(* Logix 5000 project; controller DAD143_Test0 1769-L16ER-BB1B rev 34.12; software revision 34.01 *)

TASK MainTask (continuous, watchdog 500 ms) : MainProgram

MODULES
   Local : 1769-L16ER-BB1B (PointIO 0, rev 34.12)
      DAD143_1 : vendor 1358 type 12 code 1430 (Ethernet 192.168.210.10, rev 1.4, StandardDataDriven RPI 20 ms)
      Discrete_IO : Embedded (PointIO 1, rev 34.11, Output RPI 20 ms)
END_MODULES

ADD_ON_INSTRUCTION AOI_DAD_143_Read   (* revision 1.0 *)
VAR_INPUT
   Index_0 : SINT; {visible}
   Index_1 : SINT; {visible}
   Subindex : SINT; {visible}
END_VAR
VAR_IN_OUT
   Out_Parameter : SINT[3]; {required}
END_VAR

ROUTINE Logic   (* ladder *)
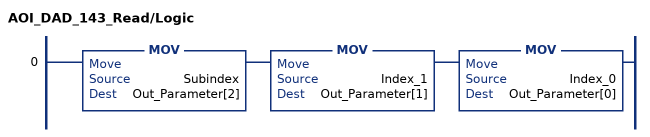
   0: MOV(Subindex,Out_Parameter[2])MOV(Index_1,Out_Parameter[1])MOV(Index_0,Out_Parameter[0]);
END_ROUTINE
END_ADD_ON_INSTRUCTION

ADD_ON_INSTRUCTION AOI_DAD_143_Write   (* revision 1.0 *)
VAR_IN_OUT
   Index_and_Subindex : SINT[3]; {required}
END_VAR
VAR_INPUT
   Data_0 : SINT; {required}
   Data_1 : SINT; {required}
   Data_2 : SINT; {required}
   Data_3 : SINT; {required}
END_VAR
VAR_IN_OUT
   Write_Par : SINT[7]; {required}
END_VAR

ROUTINE Logic   (* ladder *)
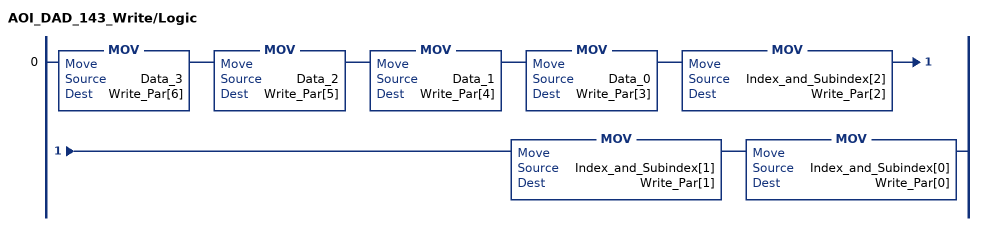
   0: MOV(Data_3,Write_Par[6])MOV(Data_2,Write_Par[5])MOV(Data_1,Write_Par[4])MOV(Data_0,Write_Par[3])MOV(Index_and_Subindex[2],Write_Par[2])MOV(Index_and_Subindex[1],Write_Par[1])MOV(Index_and_Subindex[0],Write_Par[0]);
END_ROUTINE
END_ADD_ON_INSTRUCTION

ADD_ON_INSTRUCTION AOI_DAD_143_Write_1   (* revision 1.0 *)
VAR_INPUT
   Index_0 : SINT; {visible}
   Index_1 : SINT; {visible}
   Subindex : SINT; {visible}
   Data_0 : SINT; {visible}
   Data_1 : SINT; {visible}
   Data_2 : SINT; {visible}
   Data_3 : SINT; {visible}
END_VAR
VAR_IN_OUT
   Write_Par : SINT[7]; {required}
END_VAR

ROUTINE Logic   (* ladder *)
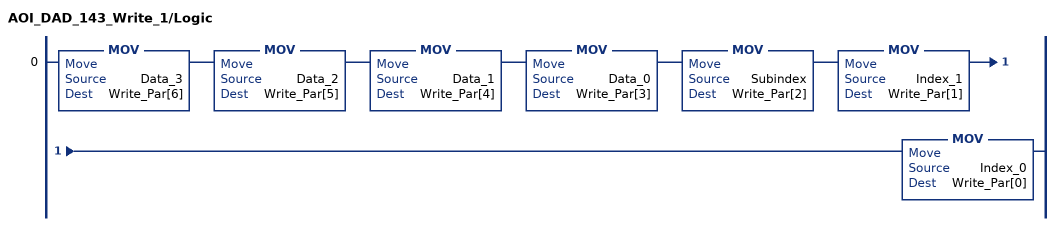
   0: MOV(Data_3,Write_Par[6])MOV(Data_2,Write_Par[5])MOV(Data_1,Write_Par[4])MOV(Data_0,Write_Par[3])MOV(Subindex,Write_Par[2])MOV(Index_1,Write_Par[1])MOV(Index_0,Write_Par[0]);
END_ROUTINE
END_ADD_ON_INSTRUCTION

VAR_GLOBAL   (* controller tags *)
   CE_Read : BOOL;
   CE_Read_Par : SINT[3];
   CE_Read_Res : SINT[5] := ([0] := 16#0b);
   CE_Read_Value : SINT := 11;
   CE_Read_Value_1 : SINT;
   CE_Read_Value_2 : SINT;
   CE_Read_Value_3 : SINT;
   CE_Start : BOOL;
   CE_Step1 : BOOL;
   CE_Step2 : BOOL;
   CE_Step3 : BOOL;
   CE_Write : BOOL;
   CI_Change : BOOL;
   CI_Change_Handshake : BOOL;
   CI_Change_Tag : BOOL;
   CI_Read_Par : SINT[3];
   CI_Step1 : BOOL;
   CI_Val : DINT;
   CM1_Change : BOOL;
   CM1_Change_Handshake : BOOL;
   CM1_Change_Tag : BOOL;
   CM1_Read_Par : SINT[3];
   CM1_Step1 : BOOL;
   CM1_Val : DINT;
   CM2_Change : BOOL;
   CM2_Change_Handshake : BOOL;
   CM2_Change_Tag : BOOL;
   CM2_Read_Par : SINT[3];
   CM2_Step1 : BOOL;
   CM2_Val : DINT;
   CM3_Change : BOOL;
   CM3_Change_Handshake : BOOL;
   CM3_Change_Tag : BOOL;
   CM3_Read_Par : SINT[3];
   CM3_Step1 : BOOL;
   CM3_Val : DINT;
   CS_Change : BOOL;
   CS_Change_Handshake : BOOL;
   CS_Change_Tag : BOOL;
   CS_Read_Par : SINT[3];
   CS_Step1 : BOOL;
   Cycle_Start : BOOL;
   DecimalPoint : SINT;
   Display_real : REAL := 7.79;
   DisplayStr : STRING := '7.82000017';
   DP : BOOL;
   DP_Cahr : STRING := '.';
   DP_Change : BOOL;
   DP_Change_1 : BOOL;
   DP_Change_Handshake : BOOL;
   DP_Change_Tag : BOOL;
   DP_Read : BOOL;
   DP_Read_Par : SINT[3];
   DP_Read_Res : SINT[5];
   DP_Step1 : BOOL;
   DP_Val : SINT;
   DP_Write : BOOL;
   DpPos : DINT := 4;
   DS : BOOL;
   DS_Change : BOOL;
   DS_Change_Handshake : BOOL;
   DS_Change_Tag : BOOL;
   DS_Read_Par : SINT[3];
   DS_Read_Res : SINT[5];
   DS_Step1 : BOOL;
   DS_Val : DINT;
   FinalStr : STRING := '7.76';
   FM_Change : BOOL;
   FM_Change_Handshake : BOOL;
   FM_Change_Tag : BOOL;
   FM_Read_Par : SINT[3];
   FM_Step1 : BOOL;
   FM_Val : SINT;
   gross : BOOL := 1;
   Gross_Display : DINT;
   Gross_weight : BOOL := 1;
   Int_reading : BOOL;
   MR : BOOL;
   MR_Change : BOOL;
   MR_Change_Handshake : BOOL;
   MR_Change_Tag : BOOL;
   MR_Read_Par : SINT[3];
   MR_Step1 : BOOL;
   MR_Val : SINT;
   ons_1 : BOOL;
   ons_2 : BOOL;
   Power_T : TIMER[12] := ([0].PRE := 50, [1].PRE := 50, [2].PRE := 2000, [3].PRE := 50);
   Power_T0 : TIMER := (PRE := 5000);
   READ_AOI : AOI_DAD_143_Read[18] := ([0].Index_1 := 16#23, [0].Subindex := 16#03, [1].Index_1 := 16#23, [1].Subindex := 16#03, [2].Index_1 := 16#23, [2].Subindex := 16#0b, [3].Index_1 := 16#23, [3].Subindex := 16#0b, [4].Index_1 := 16#23, [4].Subindex := 16#0c, [5].Index_1 := 16#23, [5].Subindex := 16#0d, [6].Index_1 := 16#23, [6].Subindex := 16#13, [7].Index_1 := 16#23, [7].Subindex := 16#15, [8].Index_0 := 16#04, [8].Index_1 := 16#20, [8].Subindex := 16#02, [9].Index_1 := 16#23, [9].Subindex := 16#14, [10].Index_1 := 16#23, [10].Subindex := 16#07, [11].Index_1 := 16#23, [11].Subindex := 16#08, [12].Index_1 := 16#23, [12].Subindex := 16#0e, [13].Index_1 := 16#23, [13].Subindex := 16#0f, [14].Index_1 := 16#23, [14].Subindex := 16#10);
   ReadCDP : MESSAGE;
        MessageParameters(ServiceCode := 16#0032, LocalElement := DP_Read_Par[0], DestinationTag := DP_Read_Res[0], ...)
   ReadCE : MESSAGE;
        MessageParameters(ServiceCode := 16#0032, LocalElement := CE_Read_Par[0], DestinationTag := CE_Read_Res[0], ...)
   ReadDS : MESSAGE;
        MessageParameters(ServiceCode := 16#0032, LocalElement := DS_Read_Par[0], DestinationTag := DS_Read_Res[0], ...)
   Stable_Bit : BOOL := 1;
   Start : BOOL;
   Start_Visibility : BOOL;
   T10 : TIMER := (PRE := 200);
   T11 : TIMER := (PRE := 50);
   T12 : TIMER := (PRE := 200);
   T13 : TIMER := (PRE := 200);
   T14 : TIMER := (PRE := 50);
   T15 : TIMER := (PRE := 200);
   T16 : TIMER := (PRE := 200);
   T17 : TIMER := (PRE := 50);
   T18 : TIMER := (PRE := 200);
   T19 : TIMER := (PRE := 200);
   T20 : TIMER := (PRE := 50);
   T21 : TIMER := (PRE := 200);
   T22 : TIMER := (PRE := 200);
   T23 : TIMER := (PRE := 50);
   T24 : TIMER := (PRE := 200);
   T25 : TIMER := (PRE := 200);
   T26 : TIMER := (PRE := 50);
   T27 : TIMER := (PRE := 200);
   T28 : TIMER := (PRE := 200);
   T29 : TIMER := (PRE := 50);
   T30 : TIMER := (PRE := 200);
   T31 : TIMER := (PRE := 200);
   T32 : TIMER := (PRE := 50);
   T33 : TIMER := (PRE := 200);
   T34 : TIMER := (PRE := 200);
   T35 : TIMER := (PRE := 50);
   T36 : TIMER := (PRE := 200);
   T37 : TIMER := (PRE := 200);
   T38 : TIMER := (PRE := 50);
   T39 : TIMER := (PRE := 200);
   T4 : TIMER := (PRE := 200);
   T5 : TIMER := (PRE := 200);
   T6 : TIMER := (PRE := 50);
   T7 : TIMER := (PRE := 200);
   T8 : TIMER := (PRE := 50);
   T9 : TIMER := (PRE := 200);
   Tare : BOOL;
   Tare_reset : BOOL;
   Tare_Reset_1 : BOOL;
   Tare_reset_Bit : BOOL := 1;
   Tare_set : BOOL;
   Tare_set_Bit : BOOL;
   temp : BOOL;
   temp1 : BOOL;
   temp_1 : BOOL;
   TN_Change : BOOL;
   TN_Change_Handshake : BOOL;
   TN_Change_Tag : BOOL;
   TN_Read_Par : SINT[3];
   TN_Step1 : BOOL;
   TN_Val : SINT;
   Write_AOI : AOI_DAD_143_Write[12];
   Write_AOI_1 : AOI_DAD_143_Write_1[20] := ([0].Index_1 := 16#23, [0].Subindex := 16#0b, [0].Data_0 := 16#03);
   Write_CE_Par : SINT[7] := ([1] := 23, [2] := 3, [3] := 11);
   Write_CE_Status : SINT[7] := ([0] := 1);
   Write_CI_Par : SINT[7];
   Write_CI_Status : SINT[7];
   Write_CM1_Par : SINT[7];
   Write_CM1_Status : SINT[7];
   Write_CM2_Par : SINT[7];
   Write_CM2_Status : SINT[7];
   Write_CM3_Par : SINT[7];
   Write_CM3_Status : SINT[7];
   Write_CS_Par : SINT[7];
   Write_CS_Status : SINT[7];
   Write_DP_Par : SINT[7];
   Write_DP_Status : SINT[7];
   Write_DS_Par : SINT[7];
   Write_DS_Status : SINT[7];
   Write_FM_Par : SINT[7];
   Write_FM_Status : SINT[7];
   Write_MR_Par : SINT[7];
   Write_MR_Status : SINT[7];
   Write_TN_Par : SINT[7];
   Write_TN_Status : SINT[7];
   Write_ZI_Par : SINT[7];
   Write_ZI_Status : SINT[7];
   Write_ZN_Par : SINT[7];
   Write_ZN_Status : SINT[7];
   WriteCE : MESSAGE;
        MessageParameters(ServiceCode := 16#0033, LocalElement := Write_CE_Par[0], DestinationTag := Write_CE_Status[0], ...)
   WriteCI : MESSAGE;
        MessageParameters(ServiceCode := 16#0033, LocalElement := Write_CI_Par[0], DestinationTag := Write_CI_Status[0], ...)
   WriteCM1 : MESSAGE;
        MessageParameters(ServiceCode := 16#0033, LocalElement := Write_CM1_Par[0], DestinationTag := Write_CM1_Status[0], ...)
   WriteCM2 : MESSAGE;
        MessageParameters(ServiceCode := 16#0033, LocalElement := Write_CM2_Par[0], DestinationTag := Write_CM2_Status[0], ...)
   WriteCM3 : MESSAGE;
        MessageParameters(ServiceCode := 16#0033, LocalElement := Write_CM3_Par[0], DestinationTag := Write_CM3_Status[0], ...)
   WriteCS : MESSAGE;
        MessageParameters(ServiceCode := 16#0033, LocalElement := Write_CS_Par[0], DestinationTag := Write_CS_Status[0], ...)
   WriteDP : MESSAGE;
        MessageParameters(ServiceCode := 16#0033, LocalElement := Write_DP_Par[0], DestinationTag := Write_DP_Status[0], ...)
   WriteDS : MESSAGE;
        MessageParameters(ServiceCode := 16#0033, LocalElement := Write_DS_Par[0], DestinationTag := Write_DS_Status[0], ...)
   WriteFM : MESSAGE;
        MessageParameters(ServiceCode := 16#0033, LocalElement := Write_FM_Par[0], DestinationTag := Write_DS_Status[0], ...)
   WriteMR : MESSAGE;
        MessageParameters(ServiceCode := 16#0033, LocalElement := Write_MR_Par[0], DestinationTag := Write_MR_Status[0], ...)
   WriteTN : MESSAGE;
        MessageParameters(ServiceCode := 16#0033, LocalElement := Write_TN_Par[0], DestinationTag := Write_TN_Status[0], ...)
   WriteZI : MESSAGE;
        MessageParameters(ServiceCode := 16#0033, LocalElement := Write_ZI_Par[0], DestinationTag := Write_ZI_Status[0], ...)
   WriteZN : MESSAGE;
        MessageParameters(ServiceCode := 16#0033, LocalElement := Write_ZN_Par[0], DestinationTag := Write_ZN_Status[0], ...)
   Zero_reset : BOOL;
   Zero_Reset_1 : BOOL;
   Zero_reset_Bit : BOOL := 1;
   Zero_set : BOOL;
   Zero_set_Bit : BOOL;
   ZI_Change : BOOL;
   ZI_Change_Handshake : BOOL;
   ZI_Change_Tag : BOOL;
   ZI_Read_Par : SINT[3];
   ZI_Step1 : BOOL;
   ZI_Val : DINT;
   ZN_Change : BOOL;
   ZN_Change_Handshake : BOOL;
   ZN_Change_Tag : BOOL;
   ZN_Read_Par : SINT[3];
   ZN_Step1 : BOOL;
   ZN_Val : SINT;
END_VAR

PROGRAM MainProgram   (* main routine MainRoutine *)
VAR
   CE_Write_Done : BOOL;
   Done_CE : BOOL;
   DP_Change_Start : BOOL;
   T0 : TIMER := (PRE := 200);
   T1 : TIMER := (PRE := 200);
   T2 : TIMER := (PRE := 200);
   T3 : TIMER := (PRE := 200);
END_VAR

ROUTINE Calibraion_Max_1   (* ladder *)
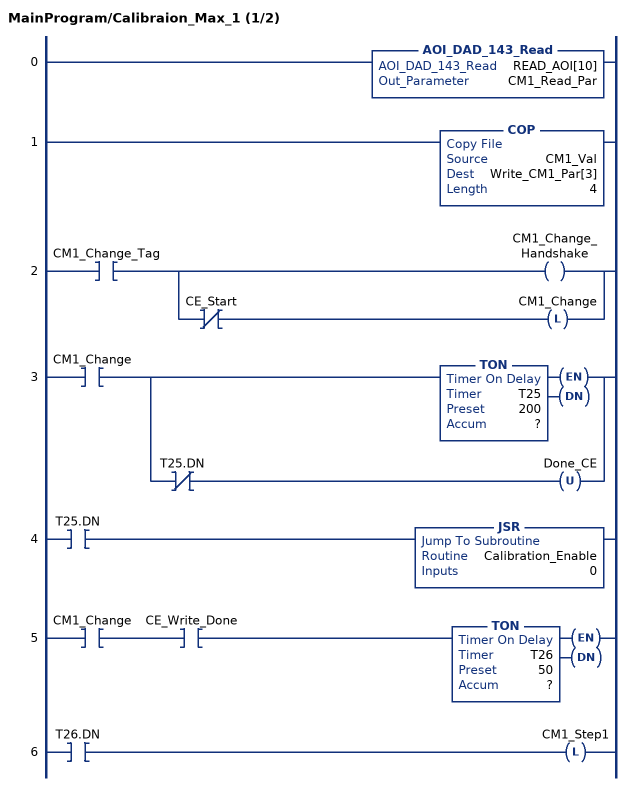
   0: AOI_DAD_143_Read(READ_AOI[10],CM1_Read_Par);
   1: COP(CM1_Val,Write_CM1_Par[3],4);
   2: XIC(CM1_Change_Tag)[OTE(CM1_Change_Handshake) ,XIO(CE_Start) OTL(CM1_Change) ];
   3: XIC(CM1_Change)[TON(T25,?,?) ,XIO(T25.DN) OTU(Done_CE) ];
   4: XIC(T25.DN)JSR(Calibration_Enable,0);
   5: XIC(CM1_Change)XIC(CE_Write_Done)TON(T26,?,?);
   6: XIC(T26.DN)OTL(CM1_Step1);
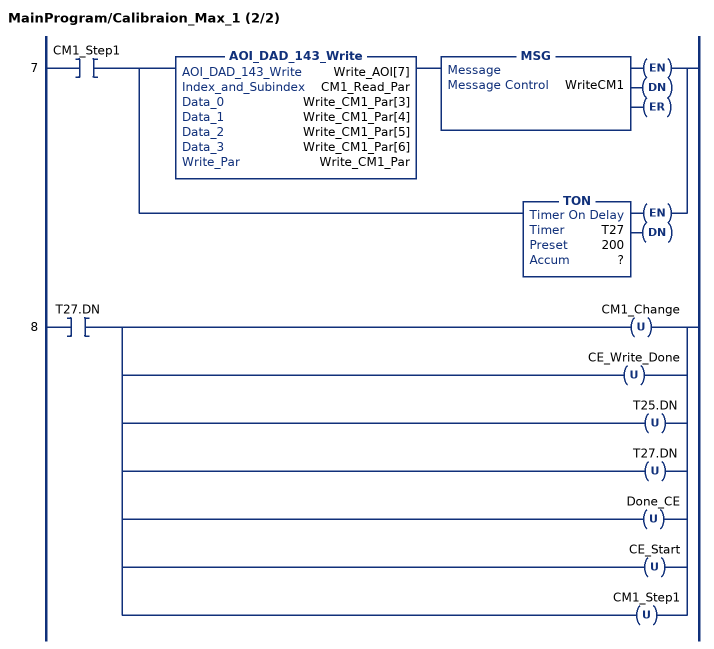
   7: XIC(CM1_Step1)[AOI_DAD_143_Write(Write_AOI[7],CM1_Read_Par,Write_CM1_Par[3],Write_CM1_Par[4],Write_CM1_Par[5],Write_CM1_Par[6],Write_CM1_Par) MSG(WriteCM1) ,TON(T27,?,?) ];
   8: XIC(T27.DN)[OTU(CM1_Change) ,OTU(CE_Write_Done) ,OTU(T25.DN) ,OTU(T27.DN) ,OTU(Done_CE) ,OTU(CE_Start) ,OTU(CM1_Step1) ];
END_ROUTINE

ROUTINE Calibraion_Max_2   (* ladder *)
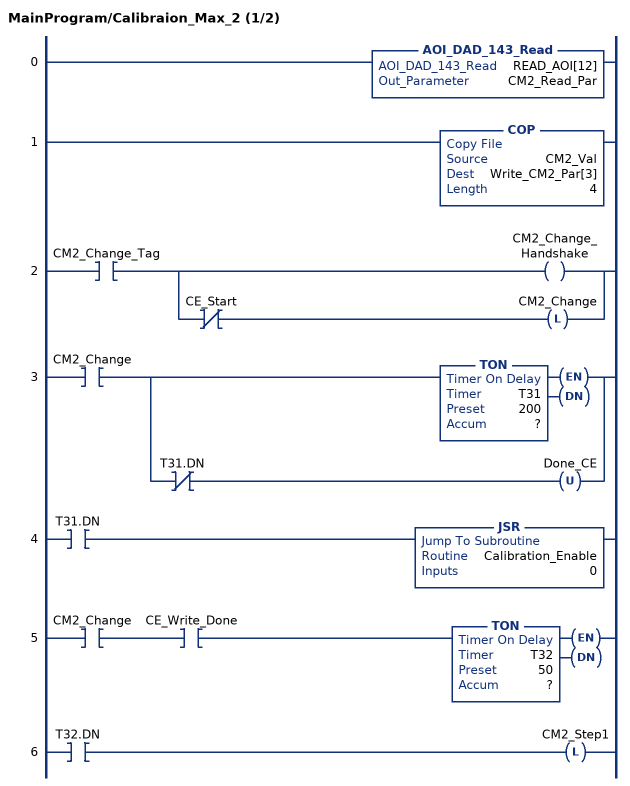
   0: AOI_DAD_143_Read(READ_AOI[12],CM2_Read_Par);
   1: COP(CM2_Val,Write_CM2_Par[3],4);
   2: XIC(CM2_Change_Tag)[OTE(CM2_Change_Handshake) ,XIO(CE_Start) OTL(CM2_Change) ];
   3: XIC(CM2_Change)[TON(T31,?,?) ,XIO(T31.DN) OTU(Done_CE) ];
   4: XIC(T31.DN)JSR(Calibration_Enable,0);
   5: XIC(CM2_Change)XIC(CE_Write_Done)TON(T32,?,?);
   6: XIC(T32.DN)OTL(CM2_Step1);
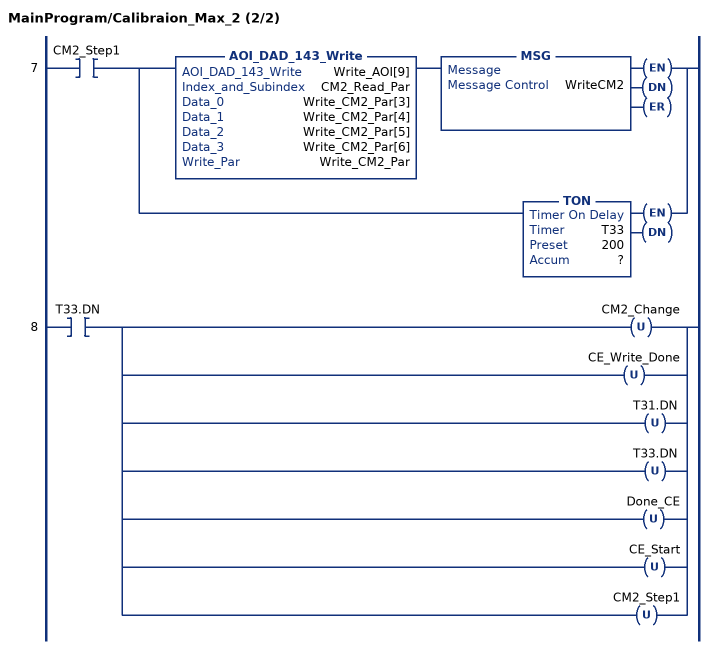
   7: XIC(CM2_Step1)[AOI_DAD_143_Write(Write_AOI[9],CM2_Read_Par,Write_CM2_Par[3],Write_CM2_Par[4],Write_CM2_Par[5],Write_CM2_Par[6],Write_CM2_Par) MSG(WriteCM2) ,TON(T33,?,?) ];
   8: XIC(T33.DN)[OTU(CM2_Change) ,OTU(CE_Write_Done) ,OTU(T31.DN) ,OTU(T33.DN) ,OTU(Done_CE) ,OTU(CE_Start) ,OTU(CM2_Step1) ];
END_ROUTINE

ROUTINE Calibraion_Max_3   (* ladder *)
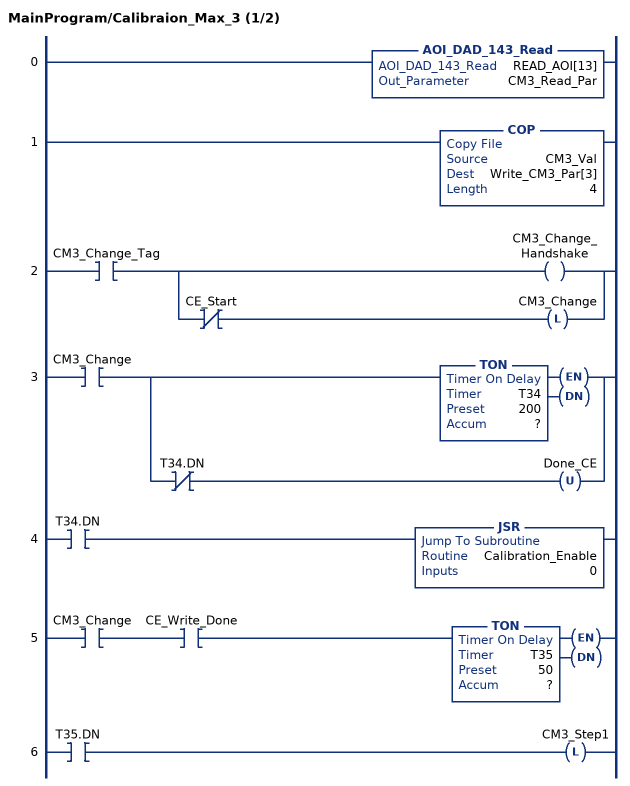
   0: AOI_DAD_143_Read(READ_AOI[13],CM3_Read_Par);
   1: COP(CM3_Val,Write_CM3_Par[3],4);
   2: XIC(CM3_Change_Tag)[OTE(CM3_Change_Handshake) ,XIO(CE_Start) OTL(CM3_Change) ];
   3: XIC(CM3_Change)[TON(T34,?,?) ,XIO(T34.DN) OTU(Done_CE) ];
   4: XIC(T34.DN)JSR(Calibration_Enable,0);
   5: XIC(CM3_Change)XIC(CE_Write_Done)TON(T35,?,?);
   6: XIC(T35.DN)OTL(CM3_Step1);
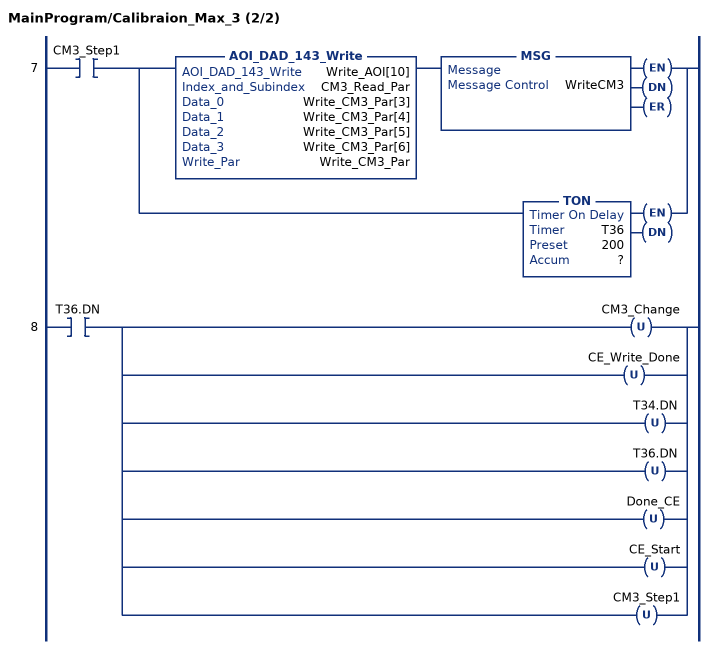
   7: XIC(CM3_Step1)[AOI_DAD_143_Write(Write_AOI[10],CM3_Read_Par,Write_CM3_Par[3],Write_CM3_Par[4],Write_CM3_Par[5],Write_CM3_Par[6],Write_CM3_Par) MSG(WriteCM3) ,TON(T36,?,?) ];
   8: XIC(T36.DN)[OTU(CM3_Change) ,OTU(CE_Write_Done) ,OTU(T34.DN) ,OTU(T36.DN) ,OTU(Done_CE) ,OTU(CE_Start) ,OTU(CM3_Step1) ];
END_ROUTINE

ROUTINE Calibration_Enable   (* ladder *)
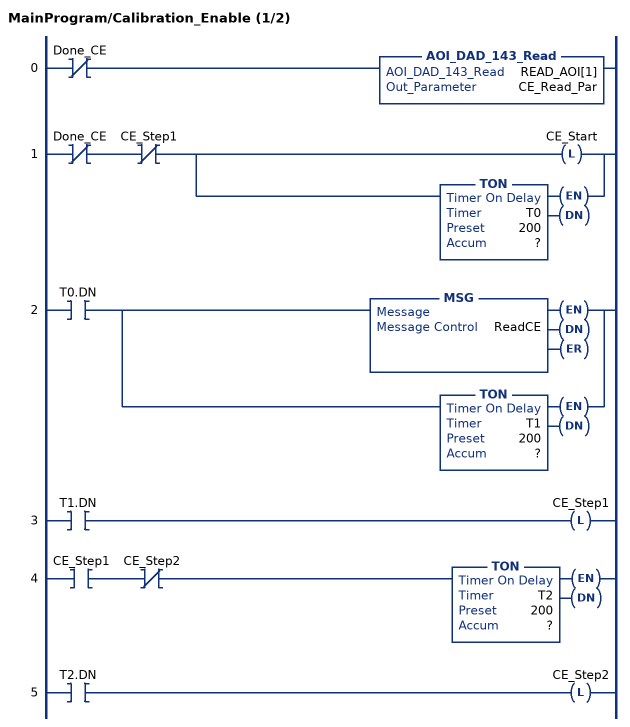
   0: XIO(Done_CE)AOI_DAD_143_Read(READ_AOI[1],CE_Read_Par);
   1: XIO(Done_CE)XIO(CE_Step1)[OTL(CE_Start) ,TON(T0,?,?) ];
   2: XIC(T0.DN)[MSG(ReadCE) ,TON(T1,?,?) ];
   3: XIC(T1.DN)OTL(CE_Step1);
   4: XIC(CE_Step1)XIO(CE_Step2)TON(T2,?,?);
   5: XIC(T2.DN)OTL(CE_Step2);
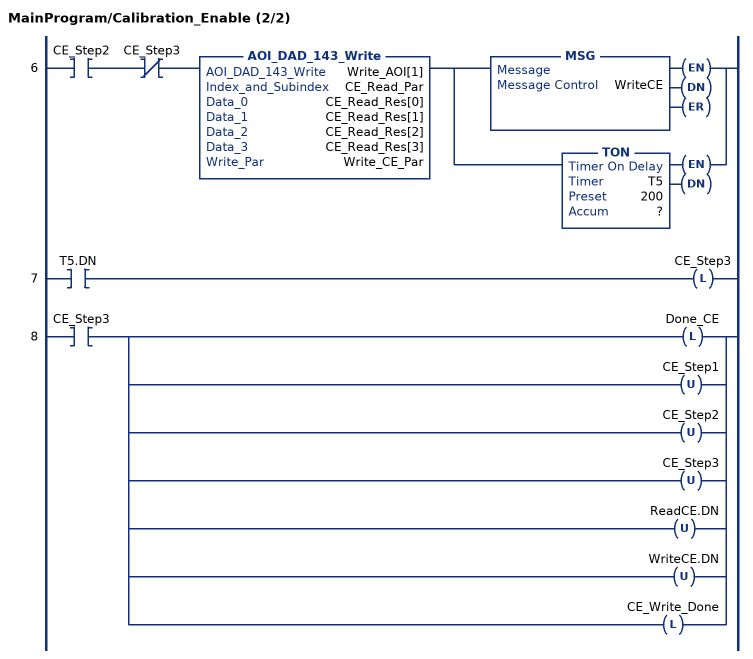
   6: XIC(CE_Step2)XIO(CE_Step3)AOI_DAD_143_Write(Write_AOI[1],CE_Read_Par,CE_Read_Res[0],CE_Read_Res[1],CE_Read_Res[2],CE_Read_Res[3],Write_CE_Par)[MSG(WriteCE) ,TON(T5,?,?) ];
   7: XIC(T5.DN)OTL(CE_Step3);
   8: XIC(CE_Step3)[OTL(Done_CE) ,OTU(CE_Step1) ,OTU(CE_Step2) ,OTU(CE_Step3) ,OTU(ReadCE.DN) ,OTU(WriteCE.DN) ,OTL(CE_Write_Done) ];
END_ROUTINE

ROUTINE Calibration_Save   (* ladder *)
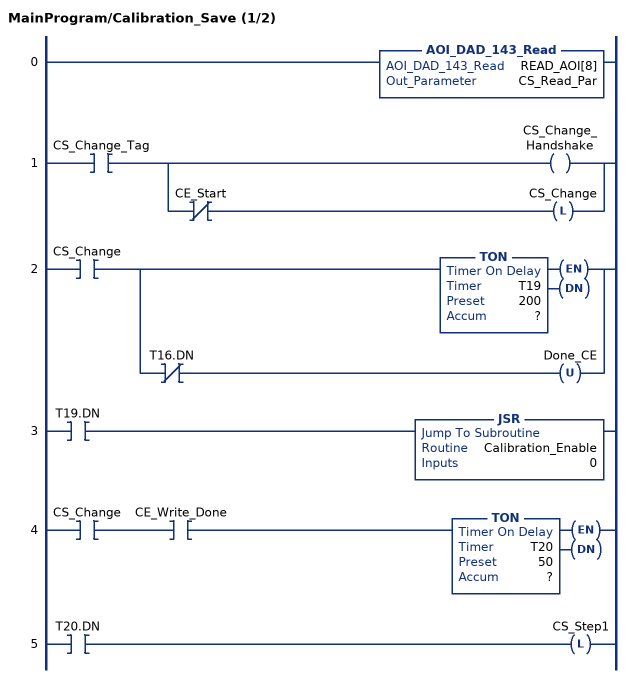
   0: AOI_DAD_143_Read(READ_AOI[8],CS_Read_Par);
   1: XIC(CS_Change_Tag)[OTE(CS_Change_Handshake) ,XIO(CE_Start) OTL(CS_Change) ];
   2: XIC(CS_Change)[TON(T19,?,?) ,XIO(T16.DN) OTU(Done_CE) ];
   3: XIC(T19.DN)JSR(Calibration_Enable,0);
   4: XIC(CS_Change)XIC(CE_Write_Done)TON(T20,?,?);
   5: XIC(T20.DN)OTL(CS_Step1);
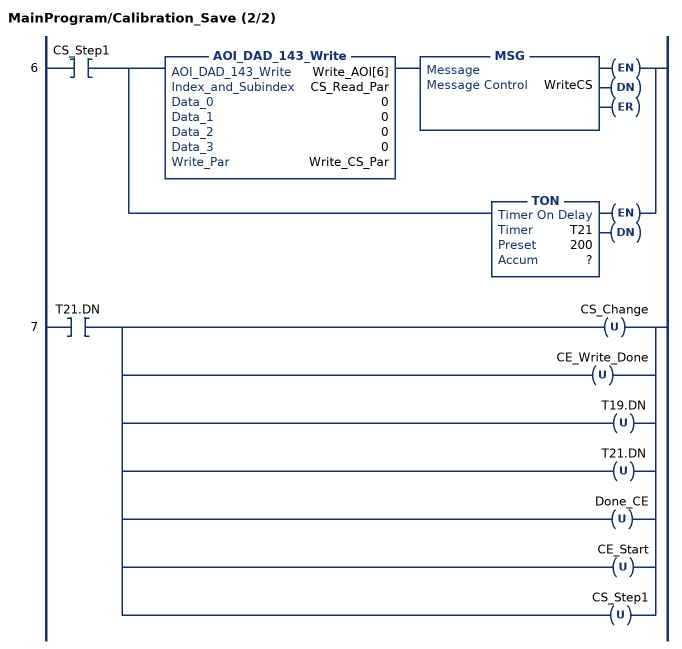
   6: XIC(CS_Step1)[AOI_DAD_143_Write(Write_AOI[6],CS_Read_Par,0,0,0,0,Write_CS_Par) MSG(WriteCS) ,TON(T21,?,?) ];
   7: XIC(T21.DN)[OTU(CS_Change) ,OTU(CE_Write_Done) ,OTU(T19.DN) ,OTU(T21.DN) ,OTU(Done_CE) ,OTU(CE_Start) ,OTU(CS_Step1) ];
END_ROUTINE

ROUTINE CI_Set_Minimum   (* ladder *)
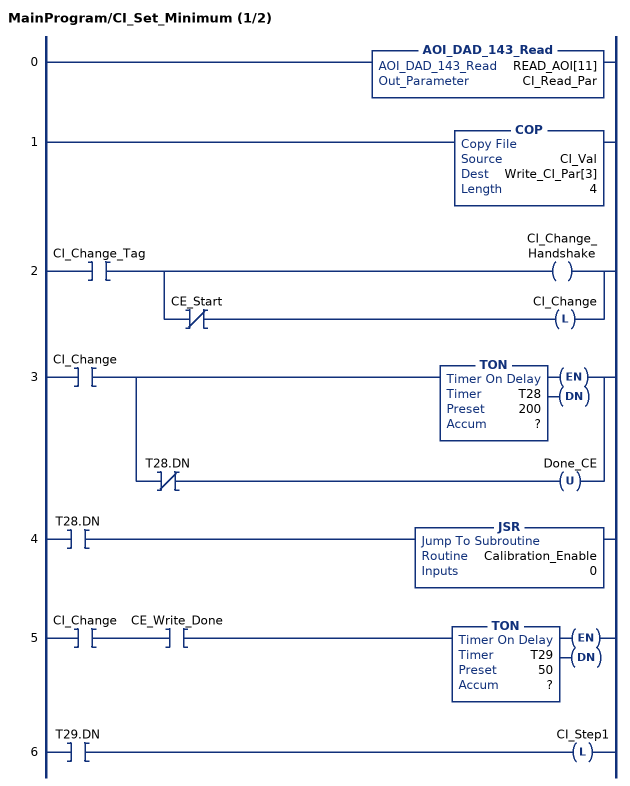
   0: AOI_DAD_143_Read(READ_AOI[11],CI_Read_Par);
   1: COP(CI_Val,Write_CI_Par[3],4);
   2: XIC(CI_Change_Tag)[OTE(CI_Change_Handshake) ,XIO(CE_Start) OTL(CI_Change) ];
   3: XIC(CI_Change)[TON(T28,?,?) ,XIO(T28.DN) OTU(Done_CE) ];
   4: XIC(T28.DN)JSR(Calibration_Enable,0);
   5: XIC(CI_Change)XIC(CE_Write_Done)TON(T29,?,?);
   6: XIC(T29.DN)OTL(CI_Step1);
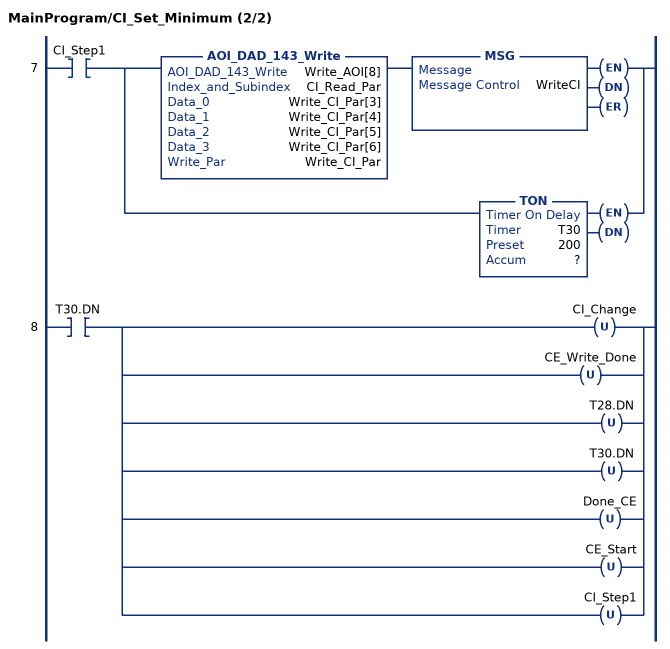
   7: XIC(CI_Step1)[AOI_DAD_143_Write(Write_AOI[8],CI_Read_Par,Write_CI_Par[3],Write_CI_Par[4],Write_CI_Par[5],Write_CI_Par[6],Write_CI_Par) MSG(WriteCI) ,TON(T30,?,?) ];
   8: XIC(T30.DN)[OTU(CI_Change) ,OTU(CE_Write_Done) ,OTU(T28.DN) ,OTU(T30.DN) ,OTU(Done_CE) ,OTU(CE_Start) ,OTU(CI_Step1) ];
END_ROUTINE

ROUTINE Decimal_Points   (* ladder *)
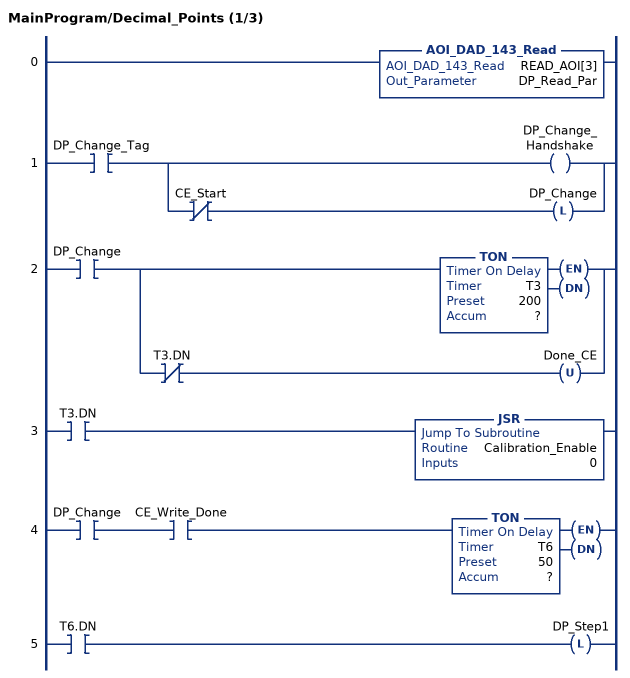
   0: AOI_DAD_143_Read(READ_AOI[3],DP_Read_Par);
   1: XIC(DP_Change_Tag)[OTE(DP_Change_Handshake) ,XIO(CE_Start) OTL(DP_Change) ];
   2: XIC(DP_Change)[TON(T3,?,?) ,XIO(T3.DN) OTU(Done_CE) ];
   3: XIC(T3.DN)JSR(Calibration_Enable,0);
   4: XIC(DP_Change)XIC(CE_Write_Done)TON(T6,?,?);
   5: XIC(T6.DN)OTL(DP_Step1);
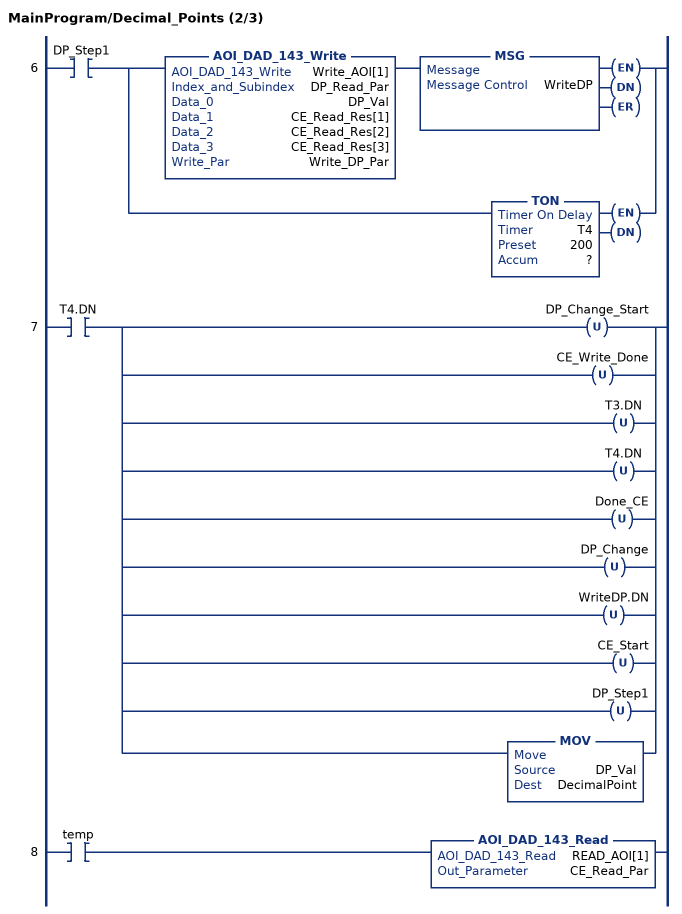
   6: XIC(DP_Step1)[AOI_DAD_143_Write(Write_AOI[1],DP_Read_Par,DP_Val,CE_Read_Res[1],CE_Read_Res[2],CE_Read_Res[3],Write_DP_Par) MSG(WriteDP) ,TON(T4,?,?) ];
   7: XIC(T4.DN)[OTU(DP_Change_Start) ,OTU(CE_Write_Done) ,OTU(T3.DN) ,OTU(T4.DN) ,OTU(Done_CE) ,OTU(DP_Change) ,OTU(WriteDP.DN) ,OTU(CE_Start) ,OTU(DP_Step1) ,MOV(DP_Val,DecimalPoint) ];
   8: XIC(temp)AOI_DAD_143_Read(READ_AOI[1],CE_Read_Par);
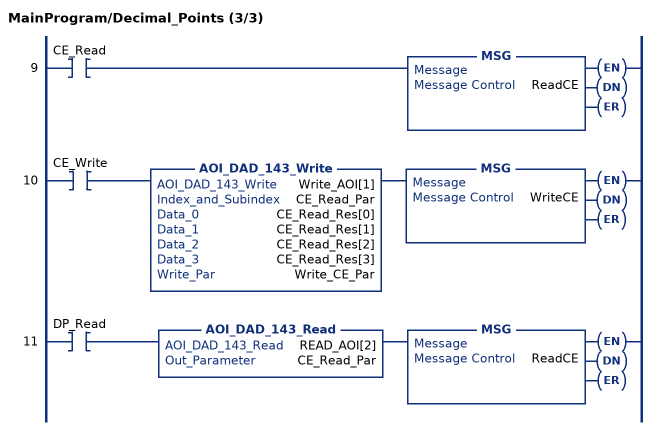
   9: XIC(CE_Read)MSG(ReadCE);
   10: XIC(CE_Write)AOI_DAD_143_Write(Write_AOI[1],CE_Read_Par,CE_Read_Res[0],CE_Read_Res[1],CE_Read_Res[2],CE_Read_Res[3],Write_CE_Par)MSG(WriteCE);
   11: XIC(DP_Read)AOI_DAD_143_Read(READ_AOI[2],CE_Read_Par)MSG(ReadCE);
END_ROUTINE
